// Mitsubishi GX Developer project: ve450_code   PLC: FX2N

PROGRAM MAIN
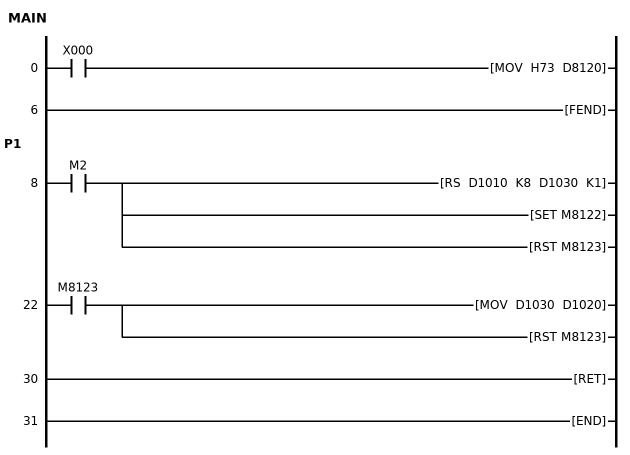
0     LD      X000
      MOV     H73 D8120
6     FEND
      P1
8     LD      M2
      RS      D1010 K8 D1030 K1
      SET     M8122
      RST     M8123
22    LD      M8123
      MOV     D1030 D1020
      RST     M8123
30    RET
31    END
END_PROGRAM

// device comments not shown above
P1  ; SEND DATA
